{attribute addProperty BoxType "EL3773-0000-0016"}
{attribute addProperty Id "U1_SAMPLESAT %I*ARRAY [1..10] OF INT16020"}
{attribute addProperty CRC "3003816138"}
{attribute addProperty SizeInBites "160"}
{attribute addProperty SizeInBytes "20"}
TYPE L1_Voltage_Samples_B30A98CA :
STRUCT
	{attribute addProperty Name "U1_SAMPLES"}
	U1_SAMPLES AT %I* : ARRAY [1..10] OF INT;
END_STRUCT
END_TYPE

(* stored: Version 1.2.0.0, ProductVersion 3.1.4024.9
   DUT L1_Voltage_Samples_B30A98CA: Id {f693d1aa-77e6-4526-aa8b-b407a8f8d87f} *)
